(* CODESYS project FunctionBlockDiagram1.project

Project tree, tasks and I/O mapping:
  Device : CODESYS Control Win V3, 3S - Smart Software Solutions GmbH, version 3.5.15.30
    application Application
      libraries: Standard, * (System)
      task MainTask (cyclic, interval t#20ms, priority 1) calls PLC_PRG, Timer_POU
      task VISU_TASK (cyclic, interval 100 ms, priority 31) calls VisuElems.Visu_Prg
      program PLC_PRG [FBD]
      visualisation Visualization
      program Timer_POU [FBD]
  text list GlobalTextList
*)

// Device/Application/PLC_PRG
PROGRAM PLC_PRG
VAR
	CTU_0: CTU;
	Contact1: BOOL := FALSE;
	Value1: WORD := 3;
	Monitor1: WORD;
	Coil1: BOOL;
	Reset1: BOOL := FALSE;
END_VAR

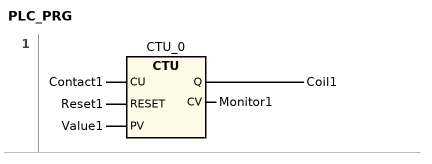
// NETWORK 1
CTU_0(CU := Contact1, RESET := Reset1, PV := Value1, CV => Monitor1); // CTU
Coil1 := CTU_0.Q;

END_PROGRAM

// Device/Application/Timer_POU
PROGRAM Timer_POU
VAR
	TON_0: TON;
	Contact1: BOOL := FALSE;
	Coil1: BOOL; (* Remember to use the ASSIGN operator to bind TON_0.Q to this *)
	CheckTime: TIME;
	EndTime: TIME := T#10S; (* Not used atm. We assign TON_0.PT as immediate *)
END_VAR

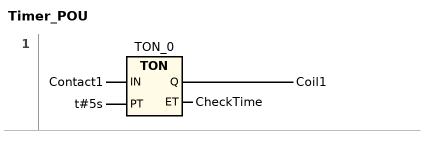
// NETWORK 1
TON_0(IN := Contact1, PT := t#5s, ET => CheckTime); // TON
Coil1 := TON_0.Q;

END_PROGRAM

// Device/Application/Visualization
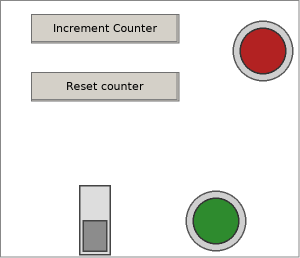
VISUALIZATION Visualization  // 300x258
    Lamp1 (228,16 70x70), variable: PLC_PRG.Coil1, style: Lamp-Lamp1-Red
    Button (31,14 148x29), "Increment Counter"
        tap PLC_PRG.Contact1
    Button (31,72 148x29), "Reset counter"
        tap PLC_PRG.Reset1
    DipSwitch (60,185 70x70), variable: Timer_POU.Contact1, behaviour: TOGGLE, style: Switch-DipSwitch-Gray
    Lamp1 (181,186 70x70), variable: Timer_POU.Coil1, style: Lamp-Lamp1-Green
END_VISUALIZATION
